{attribute 'enable_dynamic_creation'}
FUNCTION_BLOCK FB_AMR EXTENDS FB_Robot
VAR
	// AMR Properties
	jointPosition : ST_JointPosition2;
	jointVelocity : ST_JointPosition2;
	TCPPosition : ST_Pose2D;
	TCPVelocity : ST_Pose2D;
	currentGoal : ST_Target2D;
	batteryVoltage : LREAL;
	batteryLevel : INT;
	localizationPrecision : LREAL;
	isDocked : BOOL;
END_VAR

// AMR implementation

METHOD PUBLIC navigateTo : BOOL
VAR_INPUT
	goal : ST_Target2D;
END_VAR
currentGoal := goal;
// Navigate to goal
END_METHOD

METHOD PUBLIC stopNavigation : BOOL
VAR_INPUT
END_VAR
// Stop navigation
END_METHOD

METHOD PUBLIC dock : BOOL
VAR_INPUT
	dockId : INT;
END_VAR
// Dock to station
isDocked := TRUE;
END_METHOD

METHOD PUBLIC undock : BOOL
VAR_INPUT
END_VAR
// Undock from station
isDocked := FALSE;
END_METHOD

END_FUNCTION_BLOCK

(* stored: Version 1.1.0.1
   POU FB_AMR: Id {f1b2c3d4-3333-3333-3333-333333333333}
   Method navigateTo: Id {f1b2c3d4-3331-3333-3333-333333333333}
   Method stopNavigation: Id {f1b2c3d4-3332-3333-3333-333333333333}
   Method dock: Id {f1b2c3d4-3333-3333-3333-333333333333}
   Method undock: Id {f1b2c3d4-3334-3333-3333-333333333333} *)
